TYPE "FCP_STATUS_OUT"
VERSION : 0.1
// Block: FCP_STATUS_OUT
   STRUCT
      FB_Run : Bool;
      Reserved_1 : Bool;
      Reserved_2 : Bool;
      Reserved_3 : Bool;
      Mode_24V : Bool;
      Sleep_Mode : Bool;
      Converter_OK : Bool;
      Warning : Bool;
      Reserved_8 : Bool;
      Reserved_9 : Bool;
      Reserved_10 : Bool;
      Reserved_11 : Bool;
      Slave : Bool;
      ParameterGroup1 : Bool;
      Vgmin : Bool;
      Reserved_15 : Bool;
   END_STRUCT;

END_TYPE
